FUNCTION_BLOCK P_Fork (* Parallel gateway split: EI starts up to four branches at once *)
  (* Standard: 61499-2 *)
  (* Version 2.0, 2026-09-27, Project contributors, Filling cell reference model *)
  PACKAGE fillingcell;
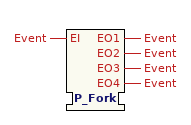
  EVENT_INPUT
    EI;
  END_EVENT
  EVENT_OUTPUT
    EO1;
    EO2;
    EO3;
    EO4;
  END_EVENT
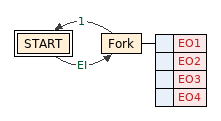
  EC_STATES
    START;
    Fork : -> EO1, -> EO2, -> EO3, -> EO4;
  END_STATES
  EC_TRANSITIONS
    START TO Fork := EI;
    Fork TO START := 1;
  END_TRANSITIONS
END_FUNCTION_BLOCK
